FUNCTION PowerFactor : REAL
VAR_INPUT
	r_P	: REAL;
	r_S	: REAL;
	r_Q	: REAL;
END_VAR

VAR
	PFRaw	: REAL;
	Factor	: INT;
END_VAR

PFRaw := ABS(r_P) / MAX(0.001, ABS(r_S));
Factor := SEL(r_Q < 0, -1, 1);

Powerfactor := LIMIT(-1, PFRaw * Factor, 1);

END_FUNCTION

(* stored: Version 1.1.0.1, ProductVersion 3.1.4026.18
   POU PowerFactor: Id {21d3fdf6-c2d9-4867-99a3-4670d4489644}, SpecialFunc None *)
